PROGRAM modbus
VAR
END_VAR

MOD_B_Local_led              :=Local_led;
MOD_B_Remote_led             :=Remote_led;
MOD_B_E_STOP_led             :=E_STOP_led;
MOD_B_Axis1_error            :=Axis1_error;
MOD_B_Axis2_error            :=Axis2_error;
MOD_B_Axis1_running          :=Axis1_running;
MOD_B_Axis2_running          :=Axis2_running;
MOD_B_Axis1_Position_done    :=Axis1_Position_done;
MOD_B_Axis2_Position_done    :=Axis2_Position_done;
MOD_B_foreward_limit_axis1_LED :=foreward_limit_axis1_LED;
MOD_B_reverse_limit_axis1_LED  :=reverse_limit_axis1_LED;
MOD_B_foreward_limit_axis2_LED :=foreward_limit_axis2_LED;
MOD_B_reverse_limit_axis2_LED  :=reverse_limit_axis2_LED;
MOB_R_Axis1_Currentvelocity  :=Axis1_Currentvelocity;
MOB_R_Axis2_Currentvelocity  :=Axis2_Currentvelocity;
MOB_R_Axis1_CurrentPosition  :=Axis1_CurrentPosition_retain;
MOB_R_Axis2_CurrentPosition  :=Axis2_CurrentPosition_retain;
MOB_R_TempController1_PV     :=TempController1_PV;
MOB_R_TempController2_PV     :=TempController2_PV;
MOB_R_LVDT1_PV               :=LVDT1_PV;
MOB_R_LVDT2_PV               :=LVDT2_PV;


IF  MOD_B_Remote_led  THEN    
	
Axis1_PositiveJog            :=MOD_B_Axis1_PositiveJog;
Axis1_NegativeJog            :=MOD_B_Axis1_NegativeJog;    
Axis1_Positionstart          :=MOD_B_Axis1_Positionstart; 
Axis1_STOP                   :=MOD_B_Axis1_STOP;
Axis2_PositiveJog            :=MOD_B_Axis2_PositiveJog;
Axis2_NegativeJog            :=MOD_B_Axis2_NegativeJog;    
Axis2_Positionstart          :=MOD_B_Axis2_Positionstart; 
Axis2_STOP                   :=MOD_B_Axis2_STOP;
MC_Reset1_Execute            :=MOD_B_MC_Reset1_Execute;
MC_Reset2_Execute            :=MOD_B_MC_Reset2_Execute;
Axis1_TargetPosition_retain  :=MOB_R_Axis1_SetPosition;
Axis2_TargetPosition_retain  :=MOB_R_Axis2_SetPosition;
Axis1_Setvelocity            :=MOB_R_Axis1_Setvelocity;
Axis2_Setvelocity            :=MOB_R_Axis2_Setvelocity;

ELSE
MOD_B_Axis1_PositiveJog       := Axis1_PositiveJog;	
MOD_B_Axis1_NegativeJog       := Axis1_NegativeJog;
MOD_B_Axis1_Positionstart     := Axis1_Positionstart;
MOD_B_Axis1_STOP              := Axis1_STOP;
MOD_B_Axis2_PositiveJog       := Axis2_PositiveJog;	
MOD_B_Axis2_NegativeJog       := Axis2_NegativeJog;
MOD_B_Axis2_Positionstart     := Axis2_Positionstart;
MOD_B_Axis2_STOP              := Axis2_STOP;
MOD_B_MC_Reset1_Execute       :=MC_Reset1_Execute;
MOD_B_MC_Reset2_Execute       :=MC_Reset2_Execute;
MOB_R_Axis1_SetPosition       :=Axis1_TargetPosition_retain;
MOB_R_Axis2_SetPosition       :=Axis2_TargetPosition_retain;
MOB_R_Axis1_Setvelocity       :=Axis1_Setvelocity;
MOB_R_Axis2_Setvelocity       :=Axis2_Setvelocity;


END_IF

END_PROGRAM

(* stored: Version 1.1.0.1, ProductVersion 3.1.4024.11
   POU modbus: Id {15ca4977-0e75-43df-9779-165aec8ec23c}, SpecialFunc None *)
